{attribute 'GeneratedUsingTerminal: KL2531-0001'}
{attribute addProperty BoxType "KL2531-0001"}
{attribute addProperty Id "Channel_1AT %Q*Channel_0D1929F00"}
{attribute addProperty CRC "1546867592"}
{attribute addProperty Size "0"}
TYPE KL_5C335388 :
STRUCT
	{attribute addProperty Name "Channel_1"}
	Channel_1 : Channel_0D1929F0;
END_STRUCT
END_TYPE

(* stored: Version 1.2.0.0, ProductVersion 3.1.4024.9
   DUT KL_5C335388: Id {dc64676e-2e16-4cea-a443-a62b4a2b90ce} *)
